// Mitsubishi GX Works2 project: servo_motor_ex7_teaching   PLC: Q02/Q02H

PROGRAM MAIN
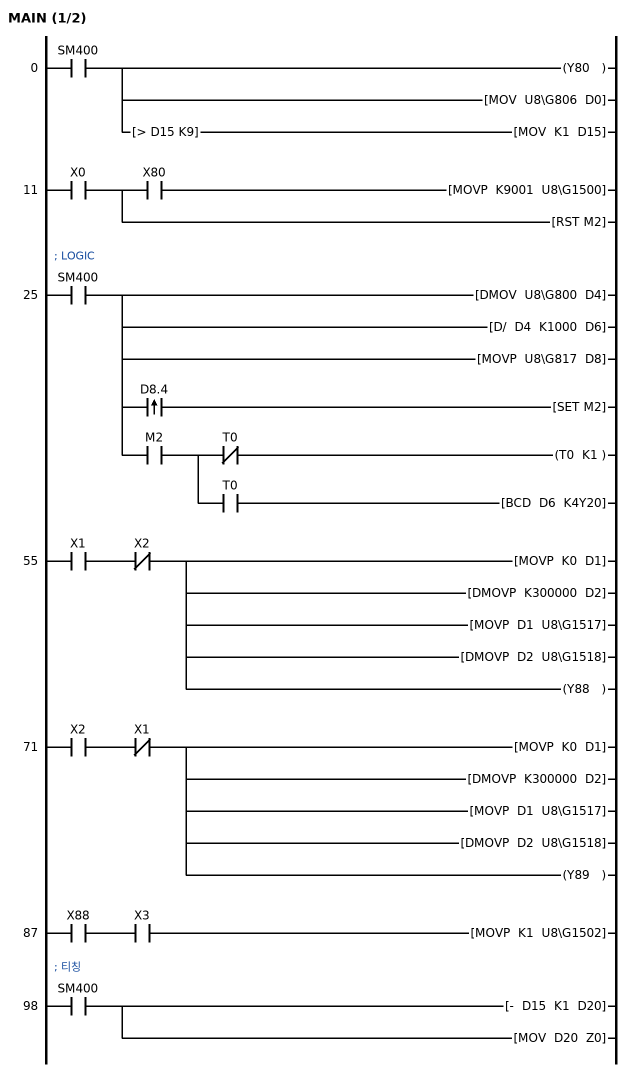
0     LD      SM400
      OUT     Y80
      MOV     U8\G806 D0
      AND>    D15 K9
      MOV     K1 D15
11    LD      X0
      MPS
      AND     X80
      MOVP    K9001 U8\G1500
      MPP
      RST     M2
; LOGIC
25    LD      SM400
      DMOV    U8\G800 D4
      D/      D4 K1000 D6
      MOVP    U8\G817 D8
      MPS
      ANDP    D8.4
      SET     M2
      MPP
      AND     M2
      MPS
      ANI     T0
      OUT     T0 K1
      MPP
      AND     T0
      BCD     D6 K4Y20
55    LD      X1
      ANI     X2
      MOVP    K0 D1
      DMOVP   K300000 D2
      MOVP    D1 U8\G1517
      DMOVP   D2 U8\G1518
      OUT     Y88
71    LD      X2
      ANI     X1
      MOVP    K0 D1
      DMOVP   K300000 D2
      MOVP    D1 U8\G1517
      DMOVP   D2 U8\G1518
      OUT     Y89
87    LD      X88
      AND     X3
      MOVP    K1 U8\G1502
; 티칭
98    LD      SM400
      -       D15 K1 D20
      MOV     D20 Z0
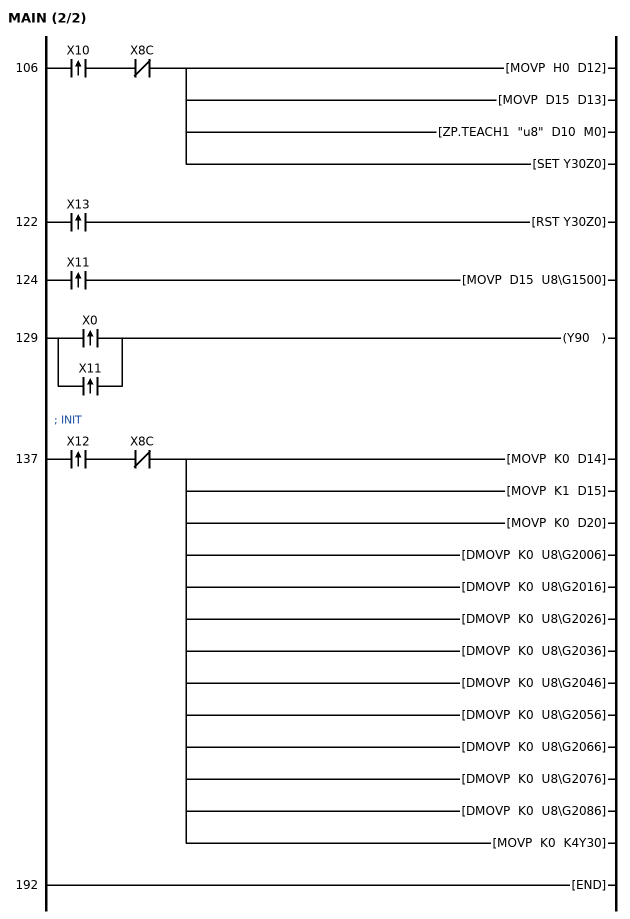
106   LDP     X10
      ANI     X8C
      MOVP    H0 D12
      MOVP    D15 D13
      ZP.TEACH1 "u8" D10 M0
      SET     Y30Z0
122   LDP     X13
      RST     Y30Z0
124   LDP     X11
      MOVP    D15 U8\G1500
129   LDP     X0
      ORP     X11
      OUT     Y90
; INIT
137   LDP     X12
      ANI     X8C
      MOVP    K0 D14
      MOVP    K1 D15
      MOVP    K0 D20
      DMOVP   K0 U8\G2006
      DMOVP   K0 U8\G2016
      DMOVP   K0 U8\G2026
      DMOVP   K0 U8\G2036
      DMOVP   K0 U8\G2046
      DMOVP   K0 U8\G2056
      DMOVP   K0 U8\G2066
      DMOVP   K0 U8\G2076
      DMOVP   K0 U8\G2086
      MOVP    K0 K4Y30
192   END
END_PROGRAM
